TYPE ST_BaseRecipeList :
STRUCT
	arrName 	: ARRAY [1..GVL_BaseConstans.MAX_NUMBER_OF_RECIPES] OF ST_BaseLabel;
	iNumber		: INT;
END_STRUCT
END_TYPE

(* stored: Version 1.1.0.1
   DUT ST_BaseRecipeList: Id {20af4396-244c-0894-2be2-65a345214b26} *)
